FUNCTION_BLOCK VALUES2ARRAY_32_BYTE (* Service Interface Function Block Type *)
  (* Description: Copyright (c) 2014 Profactor GmbH This program and the accompanying materials are made available under the terms of the Eclipse Public License 2.0 which is available at https://www.eclipse.org/legal/epl-2.0/ SPDX-License-Identifier: EPL-2.0 *)
  (* Version 3.0, 2025-04-14, Patrick Aigner, changed package *)
  (* Version 1.0, 2014-07-09, Matthias Plasch, Profactor GmbH *)
  PACKAGE eclipse4diac::convert;
  {SET_ATTRIBUTE(eclipse4diac::core::GenericClassName, 'GEN_VALUES2ARRAY')}
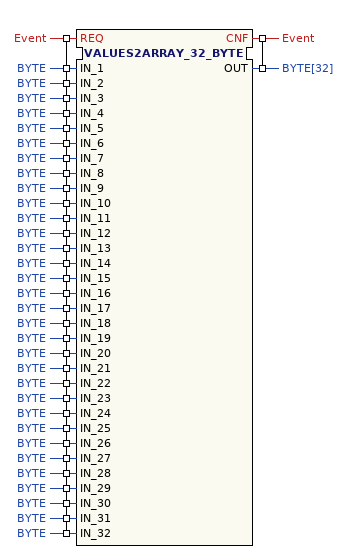
  EVENT_INPUT
    REQ WITH IN_1, IN_2, IN_3, IN_4, IN_5, IN_6, IN_7, IN_8, IN_9, IN_10, IN_11, IN_12, IN_13, IN_14, IN_15, IN_16, IN_17, IN_18, IN_19, IN_20, IN_21, IN_22, IN_23, IN_24, IN_25, IN_26, IN_27, IN_28, IN_29, IN_30, IN_31, IN_32; (* Service Request *)
  END_EVENT
  EVENT_OUTPUT
    CNF WITH OUT; (* Confirmation of Requested Service *)
  END_EVENT
  VAR_INPUT
    IN_1 : BYTE; (* input number 1 *)
    IN_2 : BYTE; (* input number 2 *)
    IN_3 : BYTE; (* input number 3 *)
    IN_4 : BYTE; (* input number 4 *)
    IN_5 : BYTE; (* input number 5 *)
    IN_6 : BYTE; (* input number 6 *)
    IN_7 : BYTE; (* input number 7 *)
    IN_8 : BYTE; (* input number 8 *)
    IN_9 : BYTE; (* input number 9 *)
    IN_10 : BYTE; (* input number 10 *)
    IN_11 : BYTE; (* input number 11 *)
    IN_12 : BYTE; (* input number 12 *)
    IN_13 : BYTE; (* input number 13 *)
    IN_14 : BYTE; (* input number 14 *)
    IN_15 : BYTE; (* input number 15 *)
    IN_16 : BYTE; (* input number 16 *)
    IN_17 : BYTE; (* input number 17 *)
    IN_18 : BYTE; (* input number 18 *)
    IN_19 : BYTE; (* input number 19 *)
    IN_20 : BYTE; (* input number 20 *)
    IN_21 : BYTE; (* input number 21 *)
    IN_22 : BYTE; (* input number 22 *)
    IN_23 : BYTE; (* input number 23 *)
    IN_24 : BYTE; (* input number 24 *)
    IN_25 : BYTE; (* input number 25 *)
    IN_26 : BYTE; (* input number 26 *)
    IN_27 : BYTE; (* input number 27 *)
    IN_28 : BYTE; (* input number 28 *)
    IN_29 : BYTE; (* input number 29 *)
    IN_30 : BYTE; (* input number 30 *)
    IN_31 : BYTE; (* input number 31 *)
    IN_32 : BYTE; (* input number 32 *)
  END_VAR
  VAR_OUTPUT
    OUT : ARRAY [0..31] OF BYTE; (* Array output *)
  END_VAR
END_FUNCTION_BLOCK
